(* PLC project ExemploPlanta.project, Vendor IEC Vendor IEC *)
(* stored: creationDateTime 2026-01-01T00:00:00 *)

FUNCTION_BLOCK FB_EXEMPLO
  VAR_INPUT
    ENTRADA : BOOL;
    TEMPO : TIME;
  END_VAR
  VAR_OUTPUT
    SAIDA_A : BOOL;
    SAIDA_B : BOOL;
  END_VAR
  VAR
    ESTADO : INT;
  END_VAR
  VAR  (* added by the conversion: wires and edge detectors of the diagram *)
    _MOVE4_ENO : BOOL;
    _MOVE4_OUT : ANY;
    _MOVE10_ENO : BOOL;
    _MOVE10_OUT : ANY;
    _EQ21_OUT : BOOL;
  END_VAR

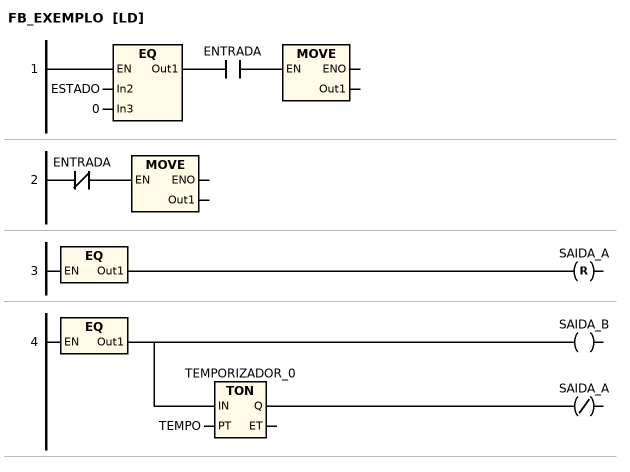
(* LD diagram, written out as Structured Text *)

_MOVE4_OUT := MOVE(EN := ESTADO = 0 AND ENTRADA, ENO => _MOVE4_ENO);
_MOVE10_OUT := MOVE(EN := NOT ENTRADA, ENO => _MOVE10_ENO);

IF EQ() THEN SAIDA_A := FALSE; END_IF;

_EQ21_OUT := EQ();
SAIDA_B := _EQ21_OUT;
TEMPORIZADOR_0(IN := _EQ21_OUT, PT := TEMPO);
SAIDA_A := NOT TEMPORIZADOR_0.Q;
END_FUNCTION_BLOCK
